Omron Sysmac Studio project CounterUP_DOWN (Sysmac Studio 1.65.0.64007, StandardProject)

# Controller new_Controller_0: NX1P2-1040DT1 version 1.69
Task PrimaryTask (priority 4, period or condition 2000): Program0

VAR_GLOBAL
    BIO_Input_Bit_00 : BOOL;  (* at BuiltInIO://cpu/#0/Input_Bit_00 *)
    BIO_Input_Bit_01 : BOOL;  (* at BuiltInIO://cpu/#0/Input_Bit_01 *)
    BIO_Input_Bit_02 : BOOL;  (* at BuiltInIO://cpu/#0/Input_Bit_02 *)
    BIO_Input_Bit_03 : BOOL;  (* at BuiltInIO://cpu/#0/Input_Bit_03 *)
    BIO_Output_Bit_00 : BOOL;  (* at BuiltInIO://cpu/#0/Output_Bit_00 *)
    IN_Start_Button : BOOL;
    IN_Stop_Button : BOOL;
    IN_OptikSensor : BOOL;
    IN_HazirButton : BOOL;
    OUT_KonveyorMotor : BOOL;
    Operator_Onay : BOOL;
    CTU1_Reset : BOOL;
    CTU1_CV : INT;
END_VAR

PROGRAM Program0
VAR
    deneme1 : BOOL;
    CTU1 : CTU;
    CTU_Reset : BOOL;
    CTU_PV : INT;
    CTU_CV : INT;
    deneme2 : BOOL;
    CTD1 : CTD;
    CTD_Load : BOOL;
    CTD_PV : INT;
    CTD_CV : INT;
    deneme3 : BOOL;
    CTUD1 : CTUD;
    CTUD_CD : BOOL;
    CTUD_Reset : BOOL;
    CTUD_Load : BOOL;
    CTUD_PV : INT;
    CTUD_QD : BOOL;
    CTUD_CV,CTD1 : INT;
    CTUD_CV : INT;
END_VAR
VAR_EXTERNAL
    BIO_Input_Bit_00 : BOOL;
    BIO_Input_Bit_01 : BOOL;
    BIO_Input_Bit_02 : BOOL;
    BIO_Input_Bit_03 : BOOL;
    IN_Start_Button : BOOL;
    IN_Stop_Button : BOOL;
    IN_OptikSensor : BOOL;
    IN_HazirButton : BOOL;
    OUT_KonveyorMotor : BOOL;
    BIO_Output_Bit_00 : BOOL;
    Operator_Onay : BOOL;
    CTU1_Reset : BOOL;
    CTU1_CV : INT;
END_VAR
VAR
    _e1 : R_TRIG;
    _e2 : R_TRIG;
    _e3 : R_TRIG;
END_VAR

(* Section Counter: ladder, written here as Structured Text *)
(* Rung 0: Konveyör Banttan her 20 koli geçtiğinde operatörün onayını bekleyen olc programını yazınız? Girişler: Start Butonu / Stop Butonu / Optik Sensör / Hazır Butonu Çıkışlar: Konveyör Motoru NOT: Sayıcı kullanarak yapınız. *)

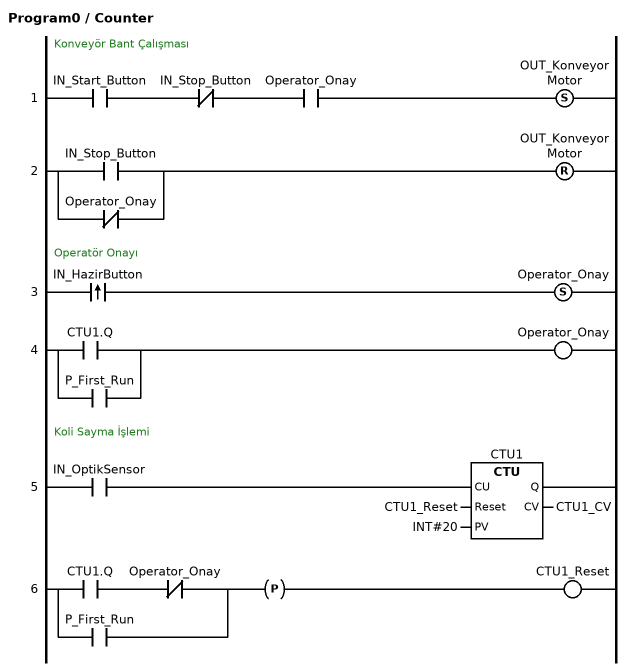
(* Rung 1: Konveyör Bant Çalışması *)
IF IN_Start_Button AND NOT IN_Stop_Button AND Operator_Onay THEN OUT_KonveyorMotor := TRUE; END_IF;
(* Rung 2 *)
IF IN_Stop_Button OR NOT Operator_Onay THEN OUT_KonveyorMotor := FALSE; END_IF;
(* Rung 3: Operatör Onayı *)
_e1(CLK := IN_HazirButton);
IF _e1.Q THEN Operator_Onay := TRUE; END_IF;
(* Rung 4 *)
Operator_Onay := CTU1.Q OR P_First_Run;
(* Rung 5: Koli Sayma İşlemi *)
_e2(CLK := IN_OptikSensor);
CTU1(CU := _e2.Q, Reset := CTU1_Reset, PV := INT#20, CV => CTU1_CV);
(* Rung 6 *)
_e3(CLK := (CTU1.Q AND NOT Operator_Onay) OR P_First_Run);
CTU1_Reset := _e3.Q;

(* Section InOut: ladder, written here as Structured Text *)

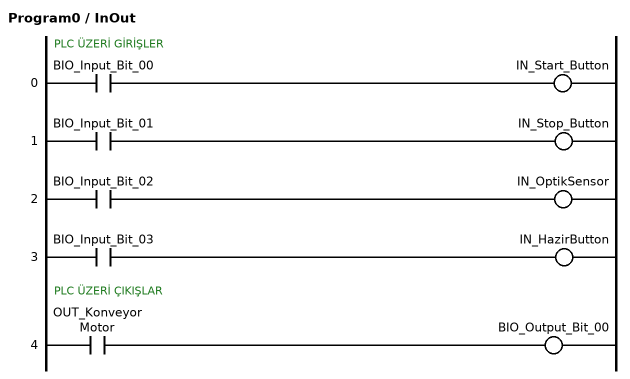
(* Rung 0: PLC ÜZERİ GİRİŞLER *)
IN_Start_Button := BIO_Input_Bit_00;
(* Rung 1 *)
IN_Stop_Button := BIO_Input_Bit_01;
(* Rung 2 *)
IN_OptikSensor := BIO_Input_Bit_02;
(* Rung 3 *)
IN_HazirButton := BIO_Input_Bit_03;
(* Rung 4: PLC ÜZERİ ÇIKIŞLAR *)
BIO_Output_Bit_00 := OUT_KonveyorMotor;
END_PROGRAM